{attribute 'qualified_only'}
TYPE PickerTokenUsage :
(
	StartToken
  ,ExecutionToken
  ,SequenceAsToken
);
END_TYPE

(* stored: Version 1.1.0.1
   DUT PickerTokenUsage: Id {1bbb9ca0-8fd7-4992-a16e-04588c8eede1} *)
